
// ===== library: MasterCopy "Cyclic interrupt PID" =====

ORGANIZATION_BLOCK "Cyclic interrupt PID"   // OB30, LAD, CyclicInterrupt
{ S7_Optimized_Access := 'TRUE' }
VERSION : 0.1
   VAR_INPUT
      Initial_Call : Bool;   // Initial call of this OB
      Event_Count : Int;   // Events discarded
   END_VAR
BEGIN

REGION Network 1
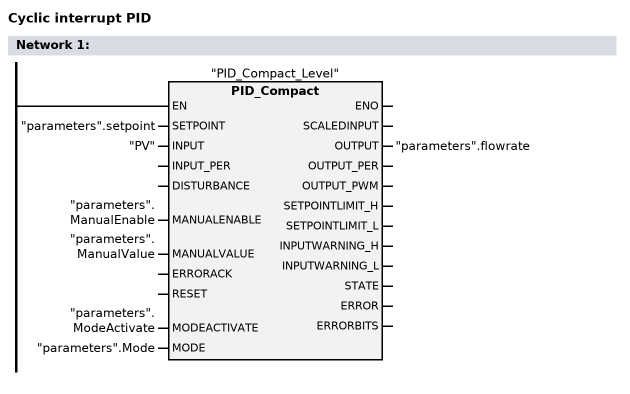
   "PID_Compact_Level"(Setpoint := "parameters".setpoint,   // PID_Compact
                       Input := "PV",
                       ManualEnable := "parameters".ManualEnable,
                       ManualValue := "parameters".ManualValue,
                       ModeActivate := "parameters".ModeActivate,
                       Mode := "parameters".Mode,
                       Output => "parameters".flowrate);
END_REGION
END_ORGANIZATION_BLOCK

// ===== library: MasterCopy "Main" =====

ORGANIZATION_BLOCK "Main"   // OB1, LAD, ProgramCycle
TITLE = "Main Program Sweep (Cycle)"
{ S7_Optimized_Access := 'TRUE' }
VERSION : 0.1
   VAR_INPUT
      Initial_Call : Bool;   // Initial call of this OB
      Remanence : Bool;   // =True, if remanent data are available
   END_VAR
BEGIN

REGION Network 1: Konnektierungsbaustein für PLC-Lab / Factory IO Function
   // Im Netzwerk 1 wird der Konnektierungsbaustein für PLC-Lab aufgerufen.
   // Dieser Aufruf darf nicht entfernt werden!
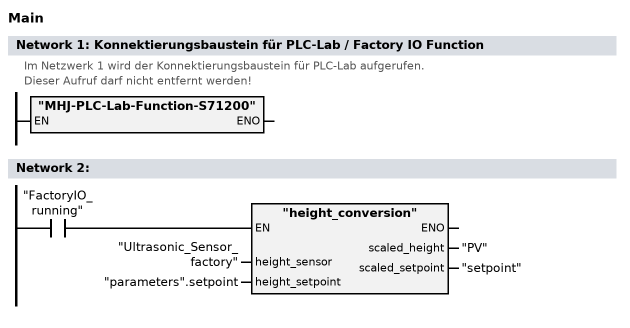
   RUNG wire#powerrail
      "MHJ-PLC-Lab-Function-S71200"()
   END_RUNG
   // the same network as SCL:
   "MHJ-PLC-Lab-Function-S71200"();
END_REGION

REGION Network 2
   RUNG wire#powerrail
      Contact( "FactoryIO_running" )
      "height_conversion"(height_sensor := "Ultrasonic_Sensor_factory", height_setpoint := "parameters".setpoint, scaled_height => "PV", scaled_setpoint => "setpoint")
   END_RUNG
   // the same network as SCL:
   IF "FactoryIO_running" THEN
       "height_conversion"(height_sensor := "Ultrasonic_Sensor_factory",
                           height_setpoint := "parameters".setpoint,
                           scaled_height => "PV",
                           scaled_setpoint => "setpoint");
   END_IF;
END_REGION
END_ORGANIZATION_BLOCK

// ===== library: MasterCopy "height_conversion" =====

FUNCTION "height_conversion" : Void   // FC1, LAD
{ S7_Optimized_Access := 'TRUE' }
VERSION : 0.1
   VAR_INPUT
      height_sensor : Real;
      height_setpoint : Int;
   END_VAR
   VAR_OUTPUT
      scaled_height : Real;
      scaled_setpoint : Real;
   END_VAR
   VAR_TEMP
      norm_height : Real;
      norm_setpoint : Real;
   END_VAR
BEGIN

REGION Network 1: Height Conversion
   // 1. Normalize the sensor output data between 0.0 and 1.0
   // 2. Scale the normalized data between minimum and maximum scale reading
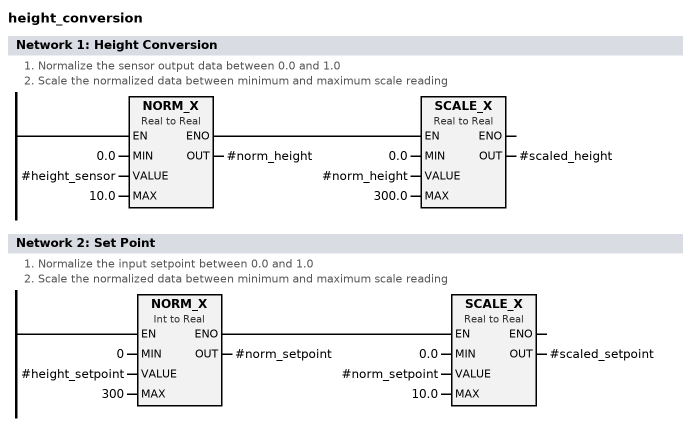
   RUNG wire#powerrail
      { S7_Templates := "[SrcType := Real, DestType := Real]" } Normalize(min := 0.0, value := #height_sensor, max := 10.0, out => #norm_height)
      { S7_Templates := "[SrcType := Real, DestType := Real]" } Scale(min := 0.0, value := #norm_height, max := 300.0, out => #scaled_height)
   END_RUNG
   // the same network as SCL:
   #norm_height := NORM_X(MIN := 0.0, VALUE := #height_sensor, MAX := 10.0);
   #scaled_height := SCALE_X(MIN := 0.0, VALUE := #norm_height, MAX := 300.0);
END_REGION

REGION Network 2: Set Point
   // 1. Normalize the input setpoint between 0.0 and 1.0
   // 2. Scale the normalized data between minimum and maximum scale reading
   RUNG wire#powerrail
      { S7_Templates := "[SrcType := Int, DestType := Real]" } Normalize(min := 0, value := #height_setpoint, max := 300, out => #norm_setpoint)
      { S7_Templates := "[SrcType := Real, DestType := Real]" } Scale(min := 0.0, value := #norm_setpoint, max := 10.0, out => #scaled_setpoint)
   END_RUNG
   // the same network as SCL:
   #norm_setpoint := NORM_X(MIN := 0, VALUE := #height_setpoint, MAX := 300);
   #scaled_setpoint := SCALE_X(MIN := 0.0, VALUE := #norm_setpoint, MAX := 10.0);
END_REGION
END_FUNCTION

// ===== library: MasterCopy "MHJ-PLC-Lab-Function-S71200" =====

FUNCTION "MHJ-PLC-Lab-Function-S71200" : Void   // FC9000, SCL
{ S7_Optimized_Access := 'TRUE' }
VERSION : 0.1
   VAR_TEMP
      rdTimeReturn : Int;
      outputTime : DTL;
      SyncVal : Byte;
      forVal : Int;
      forVal_2 : Int;
      Value : Byte;
   END_VAR
   VAR CONSTANT
      CompVal : Byte := 16#34;
      Value_01 : Byte := 16#11;
      Value_01_DW : DWord := 16#A165_D992;
      Value_02_DW : DWord := 16#58BE_4401;
   END_VAR
BEGIN

   #Value:=PEEK(area := 16#82,
        dbNumber := 0,
        byteOffset := 511);
   #Value := #Value + 1;

   POKE(area := 16#82,
        dbNumber := 0,
        byteOffset := 511,
        value := #Value);

   POKE(area:=16#81,
        dbNumber:=0,
        byteOffset:=1016,
        value:=#Value_01_DW);
   POKE(area := 16#81,
        dbNumber := 0,
        byteOffset := 1020,
        value := #Value_02_DW);

   POKE(area := 16#81,
        dbNumber := 0,
        byteOffset := 511,
        value := B#16#00);

   FOR #forVal := 0 TO 120 DO
       FOR #forVal_2:=0 TO 10 DO
           #rdTimeReturn:=RD_SYS_T(#outputTime);
           #rdTimeReturn := WR_SYS_T(#outputTime);
           #rdTimeReturn := RD_SYS_T(#outputTime);
           #rdTimeReturn := WR_SYS_T(#outputTime);
       END_FOR;
       #SyncVal:= PEEK(area := 16#81,
                      dbNumber := 0,
                      byteOffset := 511);
       IF #SyncVal = #CompVal THEN
          GOTO M_1;
       END_IF;
   END_FOR;
   RETURN;

   M_1:
   POKE(area := 16#81,
        dbNumber := 0,
        byteOffset := 511,
        value := B#16#0);
END_FUNCTION

// ===== library: MasterCopy "pump_flowrate" =====

FUNCTION "pump_flowrate" : Void   // FC2, LAD
{ S7_Optimized_Access := 'TRUE' }
VERSION : 0.1
BEGIN

REGION Network 1: flow percentage
END_REGION

REGION Network 2: flow percentage to bits
END_REGION
END_FUNCTION

// ===== library: MasterCopy "Copy of Data block in Sys_par" =====

// folder: Sys_par

DATA_BLOCK "parameters"   // DB2
{ S7_Optimized_Access := 'TRUE' }
VERSION : 0.1
   VAR
      "Process Value" : Real;
      setpoint : Int := 0;
      flowrate : Real;
      ModeActivate : Bool;
      ManualEnable : Bool;
      ManualValue : Real := 80.0;
      Mode : Int;
      Reset : Bool;
   END_VAR
BEGIN
END_DATA_BLOCK

// ===== library: MasterCopy "Inputs" =====

VAR_GLOBAL   // PLC tag table "Inputs"
   "Flow_Rate_Sensor" AT %I0.0 : Bool;
   "Float_switch_overflow" AT %I0.1 : Bool;   // S111
   "Float_switch_threshold" AT %I0.2 : Bool;   // S112
   "Low_Level_Capacitive_Sensor" AT %I0.3 : Bool;   // B114
   "High_Level_Capacitive_Sensor" AT %I0.4 : Bool;   // B113
   "Micro_switch_valve_closed" AT %I0.5 : Bool;
   "Micro_switch_valve_open" AT %I0.6 : Bool;
   "Ultrasonic_Sensor" AT %IW96 : Int;
END_VAR

// ===== library: MasterCopy "Outputs" =====

VAR_GLOBAL   // PLC tag table "Outputs"
   "Solenoid_on/off" AT %Q0.0 : Bool;
   "Heater_on/off" AT %Q0.1 : Bool;
   "Relay KF1_Pump mode" AT %Q0.2 : Bool;
   "Pump_on/off" AT %Q0.3 : Bool;
   "KF6_Proportional valve" AT %Q0.4 : Bool;
   "KF2_Fan" AT %Q0.5 : Bool;
   "Pump_P101" AT %QW96 : Int;
END_VAR

// ===== library: MasterCopy "Copy of PLC tag table in Local Tags" =====

VAR_GLOBAL   // PLC tag table "Factory tags"
   "FactoryIO_running" AT %I0.7 : Bool;
   "Ultrasonic_Sensor_factory" AT %ID30 : Real;
   "Fill valve" AT %QD30 : Real;
   "Discharge valve" AT %QD34 : Real;
   "SP" AT %QD38 : Real;
   "Flow meter" AT %ID34 : Real;
   "setpoint" AT %ID38 : Real;
   "PV" AT %QD42 : Real;
END_VAR